// TwinCAT 3 PLC project Untitled1
// ProgramVersion: 3.1.4024.0
// libraries:
//   Tc2_Standard, * (Beckhoff Automation GmbH)
//   Tc2_System, * (Beckhoff Automation GmbH)
//   Tc3_Module, * (Beckhoff Automation GmbH)
// project tree:
//   / PlcTask.TcTTO
//   POUs/ F_TrueBitsCounter.TcPOU, MAIN.TcPOU
// real-time tasks:
//   TASK PlcTask: cycle T#10ms, priority 20, ADS port 350

CONFIGURATION Untitled1
    RESOURCE PLC ON TwinCAT3
        TASK PlcTask(INTERVAL := T#10ms, PRIORITY := 20);
        PROGRAM MAIN WITH PlcTask : MAIN;
    END_RESOURCE
END_CONFIGURATION

// ---- POUs/MAIN.TcPOU
PROGRAM MAIN
VAR
	TestBitsArr		: ARRAY [0..72] OF BOOL;
	bCalc: BOOL;
	CountedTrueBits		: UINT;
	MyBitsArrSize: UINT;
END_VAR


IF bCalc THEN
	MyBitsArrSize	:= SIZEOF(TestBitsArr);
	CountedTrueBits:= F_TrueBitsCounter(pArray:= ADR(TestBitsArr),arrBitSize:= MyBitsArrSize);
	bCalc			:= FALSE;
END_IF

END_PROGRAM

// ---- POUs/F_TrueBitsCounter.TcPOU
FUNCTION F_TrueBitsCounter : UINT
VAR_INPUT
	pArray			: POINTER TO ARRAY[0..255] OF BOOL;
	arrBitSize		: UINT; 
END_VAR
	
VAR
	i				: UINT;
END_VAR



FOR i:=0 TO arrBitSize-1 DO
	IF pArray^[i] THEN
		F_TrueBitsCounter	:= F_TrueBitsCounter + 1;
	END_IF
END_FOR

END_FUNCTION
